(* IEC 61131-3 sources: rust-plc/stdlib, 4 files *)

(* ---- math.st ---- *)
(*
 * IEC 61131-3 Standard Library: Math & Selection Functions
 *
 * These are pure ST implementations of standard math and selection functions.
 *)

// ── Selection functions ──────────────────────────────────────────────

FUNCTION SEL : INT
VAR_INPUT
    G   : BOOL;   (* Selector: FALSE=IN0, TRUE=IN1 *)
    IN0 : INT;    (* Value when G=FALSE *)
    IN1 : INT;    (* Value when G=TRUE *)
END_VAR
    IF G THEN
        SEL := IN1;
    ELSE
        SEL := IN0;
    END_IF;
END_FUNCTION

FUNCTION MAX_INT : INT
VAR_INPUT
    IN1 : INT;
    IN2 : INT;
END_VAR
    IF IN1 >= IN2 THEN
        MAX_INT := IN1;
    ELSE
        MAX_INT := IN2;
    END_IF;
END_FUNCTION

FUNCTION MIN_INT : INT
VAR_INPUT
    IN1 : INT;
    IN2 : INT;
END_VAR
    IF IN1 <= IN2 THEN
        MIN_INT := IN1;
    ELSE
        MIN_INT := IN2;
    END_IF;
END_FUNCTION

FUNCTION LIMIT_INT : INT
VAR_INPUT
    MN  : INT;    (* Minimum *)
    IN1 : INT;    (* Input value *)
    MX  : INT;    (* Maximum *)
END_VAR
    IF IN1 < MN THEN
        LIMIT_INT := MN;
    ELSIF IN1 > MX THEN
        LIMIT_INT := MX;
    ELSE
        LIMIT_INT := IN1;
    END_IF;
END_FUNCTION

FUNCTION ABS_INT : INT
VAR_INPUT
    IN1 : INT;
END_VAR
    IF IN1 < 0 THEN
        ABS_INT := -IN1;
    ELSE
        ABS_INT := IN1;
    END_IF;
END_FUNCTION

// ── REAL variants ────────────────────────────────────────────────────

FUNCTION MAX_REAL : REAL
VAR_INPUT
    IN1 : REAL;
    IN2 : REAL;
END_VAR
    IF IN1 >= IN2 THEN
        MAX_REAL := IN1;
    ELSE
        MAX_REAL := IN2;
    END_IF;
END_FUNCTION

FUNCTION MIN_REAL : REAL
VAR_INPUT
    IN1 : REAL;
    IN2 : REAL;
END_VAR
    IF IN1 <= IN2 THEN
        MIN_REAL := IN1;
    ELSE
        MIN_REAL := IN2;
    END_IF;
END_FUNCTION

FUNCTION LIMIT_REAL : REAL
VAR_INPUT
    MN  : REAL;
    IN1 : REAL;
    MX  : REAL;
END_VAR
    IF IN1 < MN THEN
        LIMIT_REAL := MN;
    ELSIF IN1 > MX THEN
        LIMIT_REAL := MX;
    ELSE
        LIMIT_REAL := IN1;
    END_IF;
END_FUNCTION

FUNCTION ABS_REAL : REAL
VAR_INPUT
    IN1 : REAL;
END_VAR
    IF IN1 < 0.0 THEN
        ABS_REAL := -IN1;
    ELSE
        ABS_REAL := IN1;
    END_IF;
END_FUNCTION

(* ---- counters.st ---- *)
(*
 * IEC 61131-3 Standard Library: Counters
 *
 * CTU  — Count Up
 * CTD  — Count Down
 * CTUD — Count Up/Down
 *)

FUNCTION_BLOCK CTU
VAR_INPUT
    CU    : BOOL;   (* Count up input — counts on rising edge *)
    RESET : BOOL;   (* Reset counter to 0 *)
    PV    : INT;    (* Preset value — Q goes TRUE when CV >= PV *)
END_VAR
VAR_OUTPUT
    Q     : BOOL;   (* Output — TRUE when CV >= PV *)
    CV    : INT;    (* Current counter value *)
END_VAR
VAR
    prev_cu : BOOL := FALSE;
END_VAR
    IF RESET THEN
        CV := 0;
    ELSIF CU AND NOT prev_cu THEN
        CV := CV + 1;
    END_IF;
    prev_cu := CU;
    Q := CV >= PV;
END_FUNCTION_BLOCK

FUNCTION_BLOCK CTD
VAR_INPUT
    CD   : BOOL;   (* Count down input — counts on rising edge *)
    LOAD : BOOL;   (* Load preset value *)
    PV   : INT;    (* Preset value *)
END_VAR
VAR_OUTPUT
    Q    : BOOL;   (* Output — TRUE when CV <= 0 *)
    CV   : INT;    (* Current counter value *)
END_VAR
VAR
    prev_cd : BOOL := FALSE;
END_VAR
    IF LOAD THEN
        CV := PV;
    ELSIF CD AND NOT prev_cd THEN
        CV := CV - 1;
    END_IF;
    prev_cd := CD;
    Q := CV <= 0;
END_FUNCTION_BLOCK

FUNCTION_BLOCK CTUD
VAR_INPUT
    CU    : BOOL;   (* Count up input *)
    CD    : BOOL;   (* Count down input *)
    RESET : BOOL;   (* Reset to 0 *)
    LOAD  : BOOL;   (* Load preset value *)
    PV    : INT;    (* Preset value *)
END_VAR
VAR_OUTPUT
    QU    : BOOL;   (* Up output — TRUE when CV >= PV *)
    QD    : BOOL;   (* Down output — TRUE when CV <= 0 *)
    CV    : INT;    (* Current counter value *)
END_VAR
VAR
    prev_cu : BOOL := FALSE;
    prev_cd : BOOL := FALSE;
END_VAR
    IF RESET THEN
        CV := 0;
    ELSIF LOAD THEN
        CV := PV;
    ELSE
        IF CU AND NOT prev_cu THEN
            CV := CV + 1;
        END_IF;
        IF CD AND NOT prev_cd THEN
            CV := CV - 1;
        END_IF;
    END_IF;
    prev_cu := CU;
    prev_cd := CD;
    QU := CV >= PV;
    QD := CV <= 0;
END_FUNCTION_BLOCK

(* ---- edge_detection.st ---- *)
(*
 * IEC 61131-3 Standard Library: Edge Detection
 *
 * R_TRIG — Rising edge trigger
 * F_TRIG — Falling edge trigger
 *)

FUNCTION_BLOCK R_TRIG
VAR_INPUT
    CLK : BOOL;   (* Signal to monitor *)
END_VAR
VAR_OUTPUT
    Q   : BOOL;   (* TRUE for one cycle on rising edge *)
END_VAR
VAR
    prev : BOOL := FALSE;
END_VAR
    Q := CLK AND NOT prev;
    prev := CLK;
END_FUNCTION_BLOCK

FUNCTION_BLOCK F_TRIG
VAR_INPUT
    CLK : BOOL;   (* Signal to monitor *)
END_VAR
VAR_OUTPUT
    Q   : BOOL;   (* TRUE for one cycle on falling edge *)
END_VAR
VAR
    prev : BOOL := TRUE;
END_VAR
    Q := NOT CLK AND prev;
    prev := CLK;
END_FUNCTION_BLOCK

(* ---- timers.st ---- *)
(*
 * IEC 61131-3 Standard Library: Timers
 *
 * TON  — On-delay timer: output goes TRUE after preset time while input is TRUE
 * TOF  — Off-delay timer: output stays TRUE for preset time after input goes FALSE
 * TP   — Pulse timer: output goes TRUE for preset time on rising edge
 *
 * All timers use TIME values (milliseconds). Use TIME literals for presets:
 *   timer(IN1 := enable, PT := T#5s);     (* 5 seconds *)
 *   timer(IN1 := enable, PT := T#500ms);  (* 500 milliseconds *)
 *   timer(IN1 := enable, PT := T#1m30s);  (* 1 minute 30 seconds *)
 *
 * Timers use SYSTEM_TIME() to track wall-clock elapsed time,
 * making them independent of scan cycle speed.
 *)

FUNCTION_BLOCK TON
VAR_INPUT
    IN1  : BOOL;   (* Timer input *)
    PT   : TIME;   (* Preset time *)
END_VAR
VAR_OUTPUT
    Q    : BOOL;   (* Timer output — TRUE after PT elapsed while IN1=TRUE *)
    ET   : TIME;   (* Elapsed time *)
END_VAR
VAR
    start_time : TIME := T#0ms;
    running : BOOL := FALSE;
END_VAR
    IF IN1 THEN
        IF NOT running THEN
            running := TRUE;
            start_time := SYSTEM_TIME();
        END_IF;
        ET := SYSTEM_TIME() - start_time;
        Q := ET >= PT;
    ELSE
        running := FALSE;
        ET := T#0ms;
        Q := FALSE;
    END_IF;
END_FUNCTION_BLOCK

FUNCTION_BLOCK TOF
VAR_INPUT
    IN1  : BOOL;   (* Timer input *)
    PT   : TIME;   (* Preset time *)
END_VAR
VAR_OUTPUT
    Q    : BOOL;   (* Timer output — stays TRUE for PT after IN1 goes FALSE *)
    ET   : TIME;   (* Elapsed time *)
END_VAR
VAR
    start_time : TIME := T#0ms;
    timing : BOOL := FALSE;
END_VAR
    IF IN1 THEN
        Q := TRUE;
        ET := T#0ms;
        timing := FALSE;
    ELSE
        IF Q AND NOT timing THEN
            timing := TRUE;
            start_time := SYSTEM_TIME();
        END_IF;
        IF timing THEN
            ET := SYSTEM_TIME() - start_time;
            IF ET >= PT THEN
                Q := FALSE;
                timing := FALSE;
            END_IF;
        END_IF;
    END_IF;
END_FUNCTION_BLOCK

FUNCTION_BLOCK TP
VAR_INPUT
    IN1  : BOOL;   (* Trigger input *)
    PT   : TIME;   (* Pulse duration *)
END_VAR
VAR_OUTPUT
    Q    : BOOL;   (* Pulse output *)
    ET   : TIME;   (* Elapsed time *)
END_VAR
VAR
    start_time : TIME := T#0ms;
    pulsing  : BOOL := FALSE;
    prev_in  : BOOL := FALSE;
END_VAR
    IF IN1 AND NOT prev_in AND NOT pulsing THEN
        (* Rising edge — start pulse *)
        pulsing := TRUE;
        start_time := SYSTEM_TIME();
        Q := TRUE;
    END_IF;

    IF pulsing THEN
        ET := SYSTEM_TIME() - start_time;
        IF ET >= PT THEN
            pulsing := FALSE;
            Q := FALSE;
        END_IF;
    END_IF;

    prev_in := IN1;
END_FUNCTION_BLOCK
